// TIA Portal V18 export
DATA_BLOCK "ModeDB"   // DB2203
{ S7_Optimized_Access := 'FALSE' }
VERSION : 0.1
// stored: AutoNumber false, DBAccessibleFromOPCUA true, DBAccessibleFromWebserver true, IsOnlyStoredInLoadMemory false, IsWriteProtectedInAS false
   VAR
      Gen { S7_SetPoint := 'True'} : "ModeGenStruct";
   END_VAR
BEGIN
END_DATA_BLOCK
